// TIA Portal V16 export
// export: Created 2025-05-30T16:30:29.4413417Z, ExportSetting WithDefaults, DisplayName Totally Integrated Automation Portal, DisplayVersion V16, DisplayName TIA Portal Version Control Interface, DisplayVersion V16, DisplayName TIA Portal Openness, DisplayVersion V16, DisplayName STEP 7 Professional, DisplayVersion V16, DisplayName STEP 7 Safety, DisplayVersion V16, DisplayName WinCC Advanced, DisplayVersion V16
DATA_BLOCK "ResetOuputs_Function_Rest"   // DB29
VERSION : 0.1
// stored: AutoNumber true, InstanceOfName ResetOuputs_Function, InstanceOfType FB
"ResetOuputs_Function"
   // VAR_INPUT
   //    StopCommand_NC : Bool;
   //    StopCommand_NO : Bool;
   // END_VAR
   // VAR_OUTPUT
   //    Output_1 : Bool;
   //    Output_2 : Bool;
   //    Output_3 : Bool;
   //    Output_4 : Bool;
   //    Output_5 : Bool;
   //    Output_6 : Bool;
   //    Output_7 : Bool;
   //    Output_8 : Bool;
   //    Output_9 : Bool;
   //    Output_10 : Bool;
   // END_VAR
BEGIN
END_DATA_BLOCK
